TYPE T_CodeGTIN : STRING[20];
END_TYPE

(* stored: Version 1.1.0.1
   DUT T_CodeGTIN: Id {abbb6353-941f-487b-bb4d-e72d13c81c3c} *)
